FUNCTION_BLOCK FB_Cleaning_ValvePump EXTENDS FB_CleanDevice
VAR_INPUT
END_VAR

VAR_OUTPUT
  bO_VacuumValve                  AT %Q* : BOOL;     (*Enable vacuum valve for CleaningStation*)

  bO_VacuumPump                   AT %Q* : BOOL;     (*Enable vacuum pump for CleaningStation*)
  wO_SetPointVacuumPump           AT %Q* : WORD;     (*Vacuum pump set point*)

  bO_CleanerPump                  AT %Q* : BOOL;     (*Enable cleaner pump for CleaningStation*)
  wO_SetPointCleanerPump          AT %Q* : WORD;     (*Cleaner pump set point*)
END_VAR

VAR
  _bManuEmptyTub                         : BOOL;     (*Manually empty tub*)

  bL_VacuumValve                         : BOOL;     (*Enable vacuum valve for CleaningStation*)

  bL_VacuumPump                          : BOOL;     (*Enable vacuum pump for CleaningStation*)
  lL_SetPointVacuumPump                  : DINT;     (*Vacuum pump set point [%]*)

  bL_CleanerPump                         : BOOL;     (*Enable cleaner pump for CleaningStation*)
  lL_SetPointCleanerPump                 : DINT;     (*Cleaner pump set point [%]*)

  fb_TonCleanerPumpOffset                : TON;
  fb_TonVacuumPumpDelay                  : TON;
END_VAR

VAR PERSISTENT
  lR_AnalogMaxDigitVacuumPump            : DINT := 16383;  (*Max value analog-output in digit (32767 = 10V)*)
  lR_SetPoint1VacuumPump                 : DINT;     (*Vacuum pump set point #1 [%]*)
  lR_SetPoint2VacuumPump                 : DINT;     (*Vacuum pump set point #2 [%]*)
  lR_SetPoint3VacuumPump                 : DINT;     (*Vacuum pump set point #3 [%]*)
  lR_SetPoint4VacuumPump                 : DINT;     (*Vacuum pump set point #4 [%]*)
  lR_AnalogMaxDigitCleanerPump           : DINT := 16383;  (*Max value analog-output in digit (32767 = 10V)*)
  lR_SetPoint1CleanerPump                : DINT;     (*Cleaner pump set point #1 [%]*)
  lR_SetPoint2CleanerPump                : DINT;     (*Cleaner pump set point #2 [%]*)
  lR_SetPoint3CleanerPump                : DINT;     (*Cleaner pump set point #3 [%]*)
  lR_SetPoint4CleanerPump                : DINT;     (*Cleaner pump set point #4 [%]*)

  tR_CleanerPumpOffset                   : TIME := T#4S;
  tR_VacuumPumpDelay                     : TIME := T#1S;
  tR_VacuumPumpEmptyBin                  : TIME := T#15S;
END_VAR

METHOD mCleaning : BOOL
VAR_INPUT
  iI_Step : INT;
END_VAR
//Abort: Stop pumps and return
IF bL_AbortReq THEN
  bL_Busy        := FALSE;
  bL_Ready       := TRUE;
  bL_VacuumValve := FALSE;
  bL_VacuumPump  := FALSE;
  bL_CleanerPump := FALSE;
  mSetOutput();
  RETURN;
END_IF

//Normal operation
CASE iI_Step OF
  0: //Init - Check if axis is not activated, restore safety
    fb_TonCleanerPumpOffset(IN := FALSE, PT := tR_CleanerPumpOffset);
    fb_TonVacuumPumpDelay  (IN := FALSE, PT := tR_VacuumPumpDelay);

    bL_Busy := FALSE;

  1: //Wait for PU axis to lift
    bL_Busy := FALSE;
    
  2: //Wait for CU axis to move out
    bL_Busy := FALSE;
    
  3: //Wait for PU axis to lower
    bL_Busy := FALSE;
    
  4: //Ensure CH axis is at starting position
    bL_Busy := FALSE;

  5: //Move CH to clean start position
    bL_Busy := FALSE;

  6: //Wait until cleaning equipment ready
    bL_VacuumValve         := TRUE;

    bL_VacuumPump          := TRUE;
    lL_SetPointVacuumPump  := lR_SetPoint1VacuumPump;

    bL_CleanerPump         := TRUE;
    lL_SetPointCleanerPump := lR_SetPoint1CleanerPump;
    
    mSetOutput();

    (*Delay cleaner pump for a good start-up.*)
    fb_TonCleanerPumpOffset(IN := TRUE, PT := tR_CleanerPumpOffset);
    bL_Busy := NOT fb_TonCleanerPumpOffset.Q;
    
  7: //Cleaning
    bL_Busy := FALSE;
    
  8: //Wait until cleaning equipment ready
    bL_VacuumValve         := TRUE;

    bL_VacuumPump          := TRUE;
    lL_SetPointVacuumPump  := lR_SetPoint1VacuumPump;

    bL_CleanerPump         := FALSE;
    lL_SetPointCleanerPump := lR_SetPoint1CleanerPump;
    
    mSetOutput();

    bL_Busy := FALSE;
    
  9: //Move CH to end position
    (*Off delay vacuum pump.*)
    fb_TonVacuumPumpDelay(IN := TRUE, PT := tR_VacuumPumpDelay);
    bL_Busy := NOT fb_TonVacuumPumpDelay.Q;
    
  10: //Wait for PU axis to lift
    bL_VacuumValve := FALSE;
    bL_VacuumPump  := FALSE;
    mSetOutput();

    bL_Busy := FALSE;
    
  11: //Move CH back to start 
    bL_VacuumValve         := FALSE;

    bL_VacuumPump          := TRUE;
    lL_SetPointVacuumPump  := lR_SetPoint1VacuumPump;

    bL_CleanerPump         := FALSE;
    lL_SetPointCleanerPump := lR_SetPoint1CleanerPump;
    
    mSetOutput();

    bL_Busy := FALSE;
    
  12: //End
    bL_VacuumValve := FALSE;
    bL_VacuumPump  := FALSE;
    mSetOutput();

    bL_Busy := FALSE;
  
  ELSE
    bL_Busy := FALSE;    
END_CASE
END_METHOD

METHOD mManuSetCleanerPump
VAR_INPUT
  bI_CleanerPump                         : BOOL;     (*Enable cleaner pump for CleaningStation*)
  bI_VacuumPump                          : BOOL;     (*Enable vacuum pump for CleaningStation*)
  wI_SetPointCleanerPump                 : DINT;     (*Cleaner pump set point*)
END_VAR
IF bI_CleanerPump THEN
  bO_CleanerPump         := TRUE;
  wO_SetPointCleanerPump := DINT_TO_WORD(lR_AnalogMaxDigitCleanerPump * wI_SetPointCleanerPump / 100);

  bO_VacuumPump          := bI_VacuumPump;                                                              
  wO_SetPointVacuumPump  := DINT_TO_WORD(lR_AnalogMaxDigitVacuumPump);
ELSE
  bO_CleanerPump         := FALSE;
  bO_VacuumPump          := FALSE;
END_IF
END_METHOD

METHOD mProduction : BOOL
VAR_INPUT
  iI_Step : INT;
END_VAR
//Abort: Stop whereever axis is and return
IF bL_AbortReq THEN
  bL_Busy        := FALSE;
  bL_Ready       := TRUE;
  bL_VacuumValve := FALSE;
  bL_VacuumPump  := FALSE;
  bL_CleanerPump := FALSE;
  mSetOutput();
  RETURN;
END_IF

//Normal operation
CASE iI_Step OF
  0: //Init - Check if axis is not activated, restore safety
    fb_TonCleanerPumpOffset(IN := FALSE, PT := tR_VacuumPumpEmptyBin);

    bL_Busy := FALSE;

  1: //Wait for PU axis to lift
    bL_Busy := FALSE;
    
  2: //Wait for CU axis to move out & empty bin
    (*Timer vacuum pump to empty bin.*)
    fb_TonCleanerPumpOffset(IN := TRUE, PT := tR_VacuumPumpEmptyBin);

    bL_VacuumValve         := FALSE;

    bL_VacuumPump          := NOT fb_TonCleanerPumpOffset.Q;
    lL_SetPointVacuumPump  := lR_SetPoint1VacuumPump;

    mSetOutput();

    bL_Busy := FALSE;
    
  3: //Wait for PU axis to lower
    (*Timer vacuum pump to empty bin.*)
    fb_TonCleanerPumpOffset(IN := TRUE, PT := tR_VacuumPumpEmptyBin);

    bL_VacuumValve := FALSE;
    bL_VacuumPump  := NOT fb_TonCleanerPumpOffset.Q;
    mSetOutput();

    bL_Busy := NOT fb_TonCleanerPumpOffset.Q;
    
  4: //End
    bL_VacuumValve := FALSE;
    bL_VacuumPump  := FALSE;
    mSetOutput();

    bL_Busy := FALSE;

  ELSE
    bL_Busy := FALSE;    
END_CASE
END_METHOD

METHOD mSetOutput
VAR_INPUT
END_VAR
bO_VacuumValve         := bL_VacuumValve;

bO_VacuumPump          := bL_VacuumPump;
wO_SetPointVacuumPump  := DINT_TO_WORD(lR_AnalogMaxDigitVacuumPump * lL_SetPointVacuumPump / 100);

bO_CleanerPump         := bL_CleanerPump;
wO_SetPointCleanerPump := DINT_TO_WORD(lR_AnalogMaxDigitCleanerPump * lL_SetPointCleanerPump / 100);
END_METHOD

PROPERTY pManuEmptyTub : BOOL
GET
pManuEmptyTub := _bManuEmptyTub;
END_GET
SET
_bManuEmptyTub := pManuEmptyTub;
IF _bManuEmptyTub THEN
  bO_VacuumValve         := FALSE;
  bO_VacuumPump          := TRUE;
  wO_SetPointVacuumPump  := DINT_TO_WORD(lR_AnalogMaxDigitVacuumPump);
ELSE
  bO_VacuumValve         := FALSE;
  bO_VacuumPump          := FALSE;
END_IF
END_SET
END_PROPERTY

END_FUNCTION_BLOCK

(* stored: Version 1.1.0.1, ProductVersion 3.1.4024.9
   POU FB_Cleaning_ValvePump: Id {93b429cd-5fc8-4ec3-8be8-3b4d29fe79ec}, SpecialFunc None
   Method mCleaning: Id {e67bca71-41ea-49c8-98ca-3c4bae3c2ba5}
   Method mManuSetCleanerPump: Id {cd540726-9aa1-4443-8380-a1d258178e14}
   Method mProduction: Id {1b9d5372-e6cb-4f87-babf-3b967cf97bc5}
   Method mSetOutput: Id {435e5791-0474-450a-b952-e3ce8775febd}
   Property pManuEmptyTub: Id {28e57dd4-6351-463c-a8f9-0277f0f3c76f}
   Get Get: Id {04e83068-6c63-441a-82dd-e175fc1c371e}
   Set Set: Id {3046db68-5d58-4f53-9c4c-edffc02aed91} *)
